Fanuc KAREL source: KT00480.KL

PROGRAM KT00480
%NOLOCKGROUP
VAR
  P1: POSITION
  P2: XYZWPR
  OUT: XYZWPR
BEGIN
    P2.Y = 2.0
  OUT = P1 : P2
END KT00480
